// Mitsubishi GX Works2 project: 2016 japan robot week v2   PLC: Q03UDV

PROGRAM MAIN
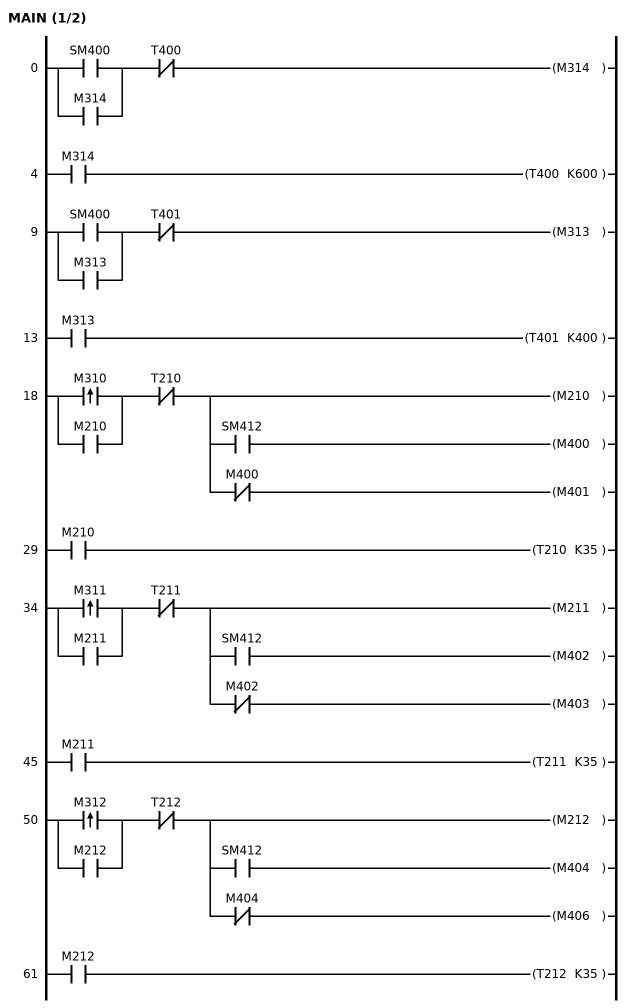
0     LD      SM400
      OR      M314
      ANI     T400
      OUT     M314
4     LD      M314
      OUT     T400 K600
9     LD      SM400
      OR      M313
      ANI     T401
      OUT     M313
13    LD      M313
      OUT     T401 K400
18    LDP     M310
      OR      M210
      ANI     T210
      OUT     M210
      MPS
      AND     SM412
      OUT     M400
      MPP
      ANI     M400
      OUT     M401
29    LD      M210
      OUT     T210 K35
34    LDP     M311
      OR      M211
      ANI     T211
      OUT     M211
      MPS
      AND     SM412
      OUT     M402
      MPP
      ANI     M402
      OUT     M403
45    LD      M211
      OUT     T211 K35
50    LDP     M312
      OR      M212
      ANI     T212
      OUT     M212
      MPS
      AND     SM412
      OUT     M404
      MPP
      ANI     M404
      OUT     M406
61    LD      M212
      OUT     T212 K35
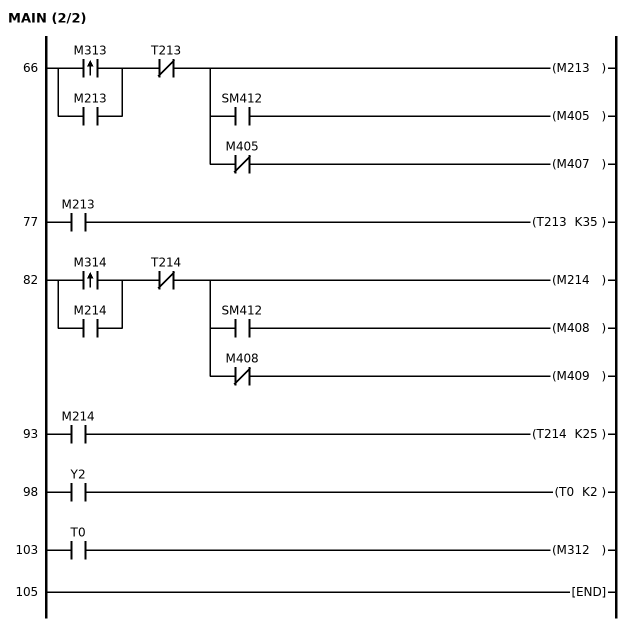
66    LDP     M313
      OR      M213
      ANI     T213
      OUT     M213
      MPS
      AND     SM412
      OUT     M405
      MPP
      ANI     M405
      OUT     M407
77    LD      M213
      OUT     T213 K35
82    LDP     M314
      OR      M214
      ANI     T214
      OUT     M214
      MPS
      AND     SM412
      OUT     M408
      MPP
      ANI     M408
      OUT     M409
93    LD      M214
      OUT     T214 K25
98    LD      Y2
      OUT     T0 K2
103   LD      T0
      OUT     M312
105   END
END_PROGRAM
